FUNCTION F_IObject_TO_IParam : I_Param
VAR_INPUT
	IObject: I_SYS_COMP_Object;
	IParam: I_Param;
END_VAR
VAR
END_VAR

__QUERYINTERFACE(IObject, IParam);
F_IObject_To_IParam := IParam;

END_FUNCTION

(* stored: Version 1.1.0.1, ProductVersion 3.1.4024.12
   POU F_IObject_TO_IParam: Id {caf6ad82-ca5a-410e-bdea-2906a70af95b}, SpecialFunc None *)
